% RSLogix 500 project conteo boton.RSS, saved by version 8.40.00.08 %
PROJECT "UNTITLED"    % processor: MicroLogix 1500 %

PROGRAM FILES
  LAD 2   4 rungs

DATA FILES
  O0 OUTPUT  4 elements
  I1 INPUT  5 elements
  S2 STATUS  66 elements
  B3 BINARY  1 elements
  T4 TIMER  1 elements
  C5 COUNTER  2 elements
  R6 CONTROL  1 elements
  N7 INTEGER  1 elements
  F8 FLOAT  1 elements

LADDER 2
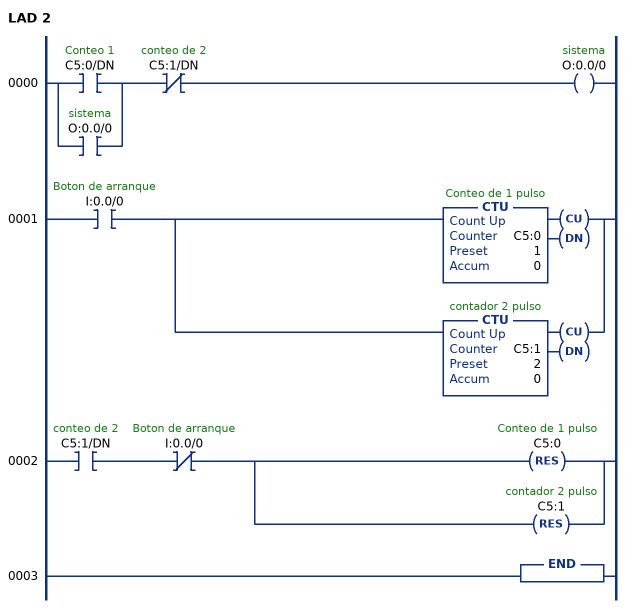
% Rung: 0 %
SOR BST XIC C5:0/DN NXB XIC O:0.0/0 BND XIO C5:1/DN OTE O:0.0/0 EOR
%   C5:0/DN  "Conteo 1" %
%   O:0.0/0  "sistema" %
%   C5:1/DN  "conteo de 2" %
% Rung: 1 %
SOR XIC I:0.0/0 BST CTU C5:0 1 0 NXB CTU C5:1 2 0 BND EOR
%   I:0.0/0  "Boton de arranque" %
%   C5:0  "Conteo de 1 pulso" %
%   C5:1  "contador 2 pulso" %
% Rung: 2 %
SOR XIC C5:1/DN XIO I:0.0/0 BST RES C5:0 NXB RES C5:1 BND EOR
%   C5:1/DN  "conteo de 2" %
%   I:0.0/0  "Boton de arranque" %
%   C5:0  "Conteo de 1 pulso" %
%   C5:1  "contador 2 pulso" %
% Rung: 3 %
SOR END EOR

DATA TABLE (non-zero values as saved)
DATA C5
% .PRE .ACC %
% C5:0 % 1 0
% C5:1 % 2 0
